FUNCTION_BLOCK ABSTRACT FB_MqttDeviceDiscoveryBase IMPLEMENTS I_MqttDeviceDiscovery
VAR_INPUT
END_VAR
VAR_OUTPUT
END_VAR
VAR
	rMqttClient : REFERENCE TO FB_IotMqttClient;
	stDeviceInformation : ST_MqttDeviceInformation;
	sNodeId : STRING(20);
	sObjectId : STRING(40);
END_VAR

PROPERTY PROTECTED ABSTRACT Component : STRING(30)
GET
END_GET
END_PROPERTY

METHOD ABSTRACT ConfigToJson : STRING(1000)
VAR_INPUT
END_VAR
END_METHOD

METHOD DeleteDevice : BOOL
VAR
	sTempTopic : STRING(255) := THIS^.DiscoveryTopic;
END_VAR
IF (__ISVALIDREF(rMqttClient)) THEN
	IF (rMqttClient.bConnected) THEN
		DeleteDevice := rMqttClient.Publish(sTopic := sTempTopic,
			pPayload := 0, nPayloadSize := 0,
			eQos := TcIotMqttQos.AtLeastOnceDelivery, bRetain := TRUE,
			bQueue := FALSE);
	END_IF
END_IF
END_METHOD

PROPERTY DeviceInformation : ST_MqttDeviceInformation
GET
DeviceInformation := this^.stDeviceInformation;
END_GET
SET
this^.stDeviceInformation := DeviceInformation;
END_SET
END_PROPERTY

METHOD PROTECTED DevInfoToJson : BOOL
VAR_INPUT
	rJsonWriter : REFERENCE TO FB_JsonSaxWriter; 
END_VAR
rJsonWriter.AddKey(key := 'dev');
rJsonWriter.StartObject();
(* setting connections is not supported at the moment... 
rJsonWriter.AddKey(key := 'cns');
rJsonWriter.StartArray();
rJsonWriter.AddString(value := stDeviceInformation.connections[0]);
rJsonWriter.AddString(value := stDeviceInformation.connections[1]);
rJsonWriter.EndArray();
*)
rJsonWriter.AddKeyString(key := 'ids', value := stDeviceInformation.identifiers);
rJsonWriter.AddKeyString(key := 'mf', value := stDeviceInformation.manufacturer);
rJsonWriter.AddKeyString(key := 'mdl', value := stDeviceInformation.model);
rJsonWriter.AddKeyString(key := 'name', value := stDeviceInformation.name);
rJsonWriter.AddKeyString(key := 'sw', value := stDeviceInformation.sw_version);
// rJsonWriter.AddKeyString(key := 'via_device', value := stDeviceInformation.via_device);
rJsonWriter.EndObject();
END_METHOD

PROPERTY PROTECTED DiscoveryTopic : STRING(255)
GET
VAR
	sTemp : STRING(255);
END_VAR
sTemp := CONCAT('homeassistant/', THIS^.Component);
sTemp := CONCAT(sTemp, '/');
sTemp := CONCAT(sTemp, THIS^.NodeId);
sTemp := CONCAT(sTemp, '/');
sTemp := CONCAT(sTemp, THIS^.ObjectId);
sTemp := CONCAT(sTemp, '/');
DiscoveryTopic := CONCAT(sTemp, 'config');
END_GET
END_PROPERTY

PROPERTY NodeId : STRING(20)
GET
NodeId := THIS^.sNodeId;
END_GET
SET
THIS^.sNodeId := NodeId;
END_SET
END_PROPERTY

PROPERTY ObjectId : STRING(40)
GET
ObjectId := THIS^.sObjectId;
END_GET
SET
THIS^.sObjectId := ObjectId;
END_SET
END_PROPERTY

METHOD RegisterDevice : BOOL
VAR
	sTempTopic : STRING(255) := THIS^.DiscoveryTopic;
	sConfig : STRING(1000) := THIS^.ConfigToJson();
END_VAR
IF (__ISVALIDREF(rMqttClient)) THEN
	IF (rMqttClient.bConnected) THEN
		RegisterDevice := rMqttClient.Publish(sTopic := sTempTopic,
			pPayload := ADR(sConfig), nPayloadSize := LEN2(ADR(sConfig)),
			eQos := TcIotMqttQos.AtLeastOnceDelivery, bRetain := TRUE,
			bQueue := FALSE);
	END_IF
END_IF
END_METHOD

METHOD PUBLIC SetMqttClient : BOOL
VAR_INPUT
	rMqttClient : REFERENCE TO FB_IotMqttClient;
END_VAR
THIS^.rMqttClient REF= rMqttClient;
END_METHOD

END_FUNCTION_BLOCK

(* stored: Version 1.1.0.1, ProductVersion 3.1.4024.5
   POU FB_MqttDeviceDiscoveryBase: Id {9654c6b2-6f10-4e61-8a0b-59ae21a32fbd}, SpecialFunc None
   Property Component: Id {3fa30243-05d8-4dad-bfc8-fb9bd082f61b}
   Get Get: Id {3b175efa-a3a6-4dbc-a88e-85f27ccc8f18}
   Method ConfigToJson: Id {a049afc8-8c59-4fa6-bc97-664fcab5cd93}
   Method DeleteDevice: Id {78be0345-afe0-4324-91af-e422264c99c9}
   Property DeviceInformation: Id {75117c2c-0749-431e-8b33-d6d3ed8cc75e}
   Get Get: Id {fafef1c8-c782-4c69-a74c-57373c47ba86}
   Set Set: Id {a016afaa-4925-40c5-9f89-a31d85a964bd}
   Method DevInfoToJson: Id {5f1e21f5-f85a-4426-bda1-29f230d1d48f}
   Property DiscoveryTopic: Id {c2d40ace-e57c-42e5-94c0-9cbf8dd81b66}
   Get Get: Id {57713942-8fe6-4a1d-8f4f-60acaf8c178f}
   Property NodeId: Id {437d477b-4be6-4f18-8bc1-e2ddaac6f988}
   Get Get: Id {94974204-25c7-42f6-bbe5-7ae587319d2b}
   Set Set: Id {3e5e9dcd-8f05-4639-8a4c-67c6e05ba21d}
   Property ObjectId: Id {d62db051-abca-4001-8368-4cf2070d2094}
   Get Get: Id {5a5e5f81-8b29-4023-852a-cb46b90eb7f1}
   Set Set: Id {31e03fae-5e7e-43d9-a262-c784cdc9a5e6}
   Method RegisterDevice: Id {3141bcb7-d277-4214-9006-27a1b29ed3e1}
   Method SetMqttClient: Id {7ee6d510-9c63-44d9-b23d-0b6b6d6df193} *)
